FUNCTION_BLOCK Test_TStreamAdd_Read_LINT EXTENDS TUnitTestBase
VAR
    Stream : TStream(StreamLength := 2);
END_VAR



Stream.Init(2);

Stream.Add_LINT(123456789);
    
Assertion.AssertEquals_UDINT(
    Expected := 8,
    Actual := Stream.Position,
    VariableName := 'Stream.Position');
    
Stream.Seek(0);

Assertion.AssertEquals_LINT(
    Expected := 123456789,
    Actual := Stream.Read_LINT(),
    VariableName := 'Stream.Read_LINT()');
    
Assertion.AssertEquals_UDINT(
    Expected := 8,
    Actual := Stream.Position,
    VariableName := 'Stream.Position');
    
    
TestFinished();

END_FUNCTION_BLOCK

(* stored: Version 1.1.0.1, ProductVersion 3.1.4024.4
   POU Test_TStreamAdd_Read_LINT: Id {d2743c81-1757-4e56-b58a-a365855abc4d}, SpecialFunc None *)
